// TwinCAT 3 PLC project FileDialog_PLC
// ProgramVersion: 3.1.4023.0
// libraries:
//   Tc2_Standard, * (Beckhoff Automation GmbH)
//   Tc2_System, * (Beckhoff Automation GmbH)
//   Tc3_Module, * (Beckhoff Automation GmbH)
// project tree:
//   DUTs/ MyStruct.TcDUT
//   GVLs/ Allgemein.TcGVL
//   / PlcTask.TcTTO
//   POUs/ MAIN.TcPOU
// real-time tasks:
//   TASK PlcTask: cycle T#10ms, priority 20, ADS port 350

CONFIGURATION FileDialog_PLC
    RESOURCE PLC ON TwinCAT3
        TASK PlcTask(INTERVAL := T#10ms, PRIORITY := 20);
        PROGRAM MAIN WITH PlcTask : MAIN;
    END_RESOURCE
END_CONFIGURATION

// ---- DUTs/MyStruct.TcDUT
TYPE MyStruct :
STRUCT
sFilePath : STRING(1024);
sFolderPath : STRING(1024);

bTriggerNewFileSelected : BOOL;
bTriggerNewFolderSelected : BOOL;
END_STRUCT
END_TYPE

// ---- GVLs/Allgemein.TcGVL
{attribute 'qualified_only'}
VAR_GLOBAL
	ImExport : MyStruct;
END_VAR

// ---- POUs/MAIN.TcPOU
PROGRAM MAIN
VAR
END_VAR

IF Allgemein.ImExport.bTriggerNewFileSelected THEN
	Allgemein.ImExport.bTriggerNewFileSelected := FALSE;
END_IF

IF Allgemein.ImExport.bTriggerNewFolderSelected THEN
	Allgemein.ImExport.bTriggerNewFolderSelected := FALSE;
END_IF

END_PROGRAM
